(*
SPDX-FileCopyrightText: © 2026 Oleksandr Tiutyk <trofimich@gmail.com>
SPDX-License-Identifier: MIT
License: https://opensource.org/license/mit
*)

(*!
<summary>Reports that a fixed-capacity collection cannot accept another element.</summary>
<description>
The caller detects the condition; this exception does not inspect or modify the collection or destination.
Uses the GeneralException task-local cycle lifetime and throw rules.
</description>
*)
INTERFACE IStaticCollectionFullException EXTENDS IGeneralException

(*!
<summary>Builds the diagnostic and raises this exception through GeneralException.</summary>
<description>
Copies the supplied diagnostic data, sets error code to zero and supplies no inner exception. Call only in a
cyclic task, not during FB_init. The caller must already have detected the reported condition.
</description>
<param name="collectionName">Collection name used in the diagnostic.</param>
<param name="capacity">Maximum number of elements, not a byte size.</param>
*)
METHOD Throw
VAR_INPUT
	sourceNamespaceName : STRING;
	sourceClassName : STRING;
	sourcePOUName : STRING;
	sourcePosition : STRING;
	collectionName : WSTRING;
	capacity : UDINT;
END_VAR
END_METHOD

END_INTERFACE

(* stored: Version 1.1.0.1
   Itf IStaticCollectionFullException: Id {dab6c626-d4d0-424f-8f97-94d7f340ac50}
   Method Throw: Id {1d5e094d-8546-408b-a259-af06e6c60cb7} *)
